// Program sprawdzajacy liczbe przekroczen czasu cyklu Task'a
PROGRAM P_PlcTaskSystemInfo
VAR_INPUT
	bReset								: BOOL;
END_VAR
VAR
	fbGetCurTaskIdx  					: GETCURTASKINDEX;
	bCycleTimeExeeded					: BOOL;
	rCounterCycleTimeExeeded			: REAL;
	rtCounterCycleTimeExeeded			: R_TRIG;
	rtReset								: R_TRIG;
	rtError								: R_TRIG;
	tonDelayAfterPowerOn: TON;
	bPowerOnDelay: BOOL;
END_VAR
VAR_OUTPUT
	bError								: BOOL;
	bOK									: BOOL;
	bWarning							: BOOL;
	udiErrorID							: UDINT;
	sErrorDescription					: WSTRING;
END_VAR

fbGetCurTaskIdx();
bCycleTimeExeeded 						:= _TaskInfo[fbGetCurTaskIdx.index].CycleTimeExceeded;

(*Dodane opóżnienie zliczania błędu po uruchomieniu maszyny*)
tonDelayAfterPowerOn					(IN:=NOT bPowerOnDelay,	PT:=T#5S);
IF tonDelayAfterPowerOn.Q THEN
	bPowerOnDelay	:=	TRUE;
END_IF

rtCounterCycleTimeExeeded				(CLK:= bCycleTimeExeeded AND bPowerOnDelay);
rtReset									(CLK:= bReset);

IF rtCounterCycleTimeExeeded.Q THEN
	rCounterCycleTimeExeeded			:= rCounterCycleTimeExeeded + 1;
END_IF	

IF rtReset.Q THEN
	rCounterCycleTimeExeeded 			:= 0;
END_IF

IF rCounterCycleTimeExeeded = 0 THEN
	P_PlcTaskSystemInfo.bError			:= FALSE;
	P_PlcTaskSystemInfo.bOK				:= TRUE;
END_IF

IF rCounterCycleTimeExeeded > 0 THEN
	P_PlcTaskSystemInfo.bError			:= TRUE;
	P_PlcTaskSystemInfo.bOK				:= FALSE;
END_IF


rtError									(CLK:= bError);

IF rtError.Q THEN
	udiErrorID							:= 91;                         
	sErrorDescription					:= "Błąd sterownika | Przekroczenie czasu cyklu";	
END_IF

IF NOT bError THEN
	udiErrorID							:= 0;	
	sErrorDescription					:= "";
END_IF

END_PROGRAM

(* stored: Version 1.1.0.1, ProductVersion 3.1.4026.13, FileIdentifier 012997db19ada9daebf87aac3b74d7af0f4aa70c, FileSignature 5357ee28293fbb1353c01ba5b8659c913c9457dc17f6fae09798f82da1abc00ab69913530bb7ec21ffe2ec14a26f27b1d9193e19a97e7efc8d9e94c462055a30f86eece4b0142550ec233d8f399903ac2c46aea0c56f0fe48a3a141000ee19ab71e4bc583dca87a8edfb66ab4fbf29836f4a329c7948511c4453527a674c078f6b462861f6e55a3d4f10cd62a0b48d4a2959e99e9b46d961371816cb3da742bbc98df50ba1473985d9f57b3ce138e90ca2d60da502177ac743bfb14b966316eb0ebafc8f1a4b2a9ce939790af5238082233aca6a2878afc23e645790f11bb67366957adc8174469bcc5ece4740ae40f9cb4ba384d09918b60cee41c03938a592
   POU P_PlcTaskSystemInfo: Id {158a92a2-9d35-4ecf-bfb2-3ecdcbfb5e15}, SpecialFunc None *)
